// TIA Portal V18 export
// export: Created 2026-01-09T11:31:58.4430527Z, ExportSetting WithDefaults, DisplayName Totally Integrated Automation Portal, DisplayVersion V18 Update 5, DisplayName TIA Portal Openness, DisplayVersion V18 Update 5, DisplayName TIA Portal Teamcenter Gateway, DisplayVersion V18, DisplayName TIA Portal Version Control Interface, DisplayVersion V18, DisplayName SINAMICS Startdrive Advanced, DisplayVersion V18 SP2 Update 1, DisplayName SINAMICS Startdrive G110M, G120, G120C, G120D, G120P, G115D, DisplayVersion V18 SP2 Update 1, DisplayName SINAMICS Startdrive G130, G150, S120, S150, SINAMICS MV, S210, G220, S200, DisplayVersion V18 SP2 Update 1, DisplayName STEP 7 Professional, DisplayVersion V18 Update 5, DisplayName STEP 7 Safety, DisplayVersion V18, DisplayName WinCC Professional, DisplayVersion V18 Update 5
TagTable "HMI_Tool"
  ST10_RecipeDB_HMI_ParameterElement_R1GripperFixtureCode : Array [0..6] of String  (PLC tag ST10_RecipeDB_HMI.ParameterElement.R1GripperFixtureCode, CPU S71500-2PN_TP700, 1 s)
    TagArrayMember "[0]"
    TagArrayMember "[1]"
    TagArrayMember "[2]"
    TagArrayMember "[3]"
    TagArrayMember "[4]"
    TagArrayMember "[5]"
    TagArrayMember "[6]"
  ST10_RecipeDB_HMI_ParameterElement_R2GripperFixtureCode : Array [0..6] of String  (PLC tag ST10_RecipeDB_HMI.ParameterElement.R2GripperFixtureCode, CPU S71500-2PN_TP700, 1 s)
    TagArrayMember "[0]"
    TagArrayMember "[1]"
    TagArrayMember "[2]"
    TagArrayMember "[3]"
    TagArrayMember "[4]"
    TagArrayMember "[5]"
    TagArrayMember "[6]"
  ST10_RecipeDB_HMI_ParameterElement_R3GripperFixtureCode : Array [0..6] of String  (PLC tag ST10_RecipeDB_HMI.ParameterElement.R3GripperFixtureCode, CPU S71500-2PN_TP700, 1 s)
    TagArrayMember "[0]"
    TagArrayMember "[1]"
    TagArrayMember "[2]"
    TagArrayMember "[3]"
    TagArrayMember "[4]"
    TagArrayMember "[5]"
    TagArrayMember "[6]"
  ST10_RecipeDB_HMI_ParameterElement_A1RingUnloadingFixtureCode : String  (PLC tag ST10_RecipeDB_HMI.ParameterElement.A1RingUnloadingFixtureCode, CPU S71500-2PN_TP700, 1 s)
  ST10_RecipeDB_HMI_ParameterElement_E1LoadingNGFixtureCode : String  (PLC tag ST10_RecipeDB_HMI.ParameterElement.E1LoadingNGFixtureCode, CPU S71500-2PN_TP700, 1 s)
  ST10_RecipeDB_HMI_ParameterElement_ShaftScanFixtureCode : String  (PLC tag ST10_RecipeDB_HMI.ParameterElement.ShaftScanFixtureCode, CPU S71500-2PN_TP700, 1 s)
  ST10_RecipeDB_HMI_ParameterElement_B1PressFixtureCode : String  (PLC tag ST10_RecipeDB_HMI.ParameterElement.B1PressFixtureCode, CPU S71500-2PN_TP700, 1 s)
  ST10_RecipeDB_HMI_ParameterElement_CGlueFixtureCode : String  (PLC tag ST10_RecipeDB_HMI.ParameterElement.CGlueFixtureCode, CPU S71500-2PN_TP700, 1 s)
  ST10_RecipeDB_HMI_ParameterElement_B1PressCylFixtureCode : String  (PLC tag ST10_RecipeDB_HMI.ParameterElement.B1PressCylFixtureCode, CPU S71500-2PN_TP700, 1 s)
  ST10_RecipeDB_HMI_ParameterElement_A2RingUnloadingFixtureCode : String  (PLC tag ST10_RecipeDB_HMI.ParameterElement.A2RingUnloadingFixtureCode, CPU S71500-2PN_TP700, 1 s)
  ST10_RecipeDB_HMI_ParameterElement_E2UnloadingNGFixtureCode : String  (PLC tag ST10_RecipeDB_HMI.ParameterElement.E2UnloadingNGFixtureCode, CPU S71500-2PN_TP700, 1 s)
  ST10_RecipeDB_HMI_ParameterElement_B2PressFixtureCode : String  (PLC tag ST10_RecipeDB_HMI.ParameterElement.B2PressFixtureCode, CPU S71500-2PN_TP700, 1 s)
  ST10_RecipeDB_HMI_ParameterElement_CGlueNGFixtureCode : String  (PLC tag ST10_RecipeDB_HMI.ParameterElement.CGlueNGFixtureCode, CPU S71500-2PN_TP700, 1 s)
  ST10_RecipeDB_HMI_ParameterElement_B2PressCylFixtureCode : String  (PLC tag ST10_RecipeDB_HMI.ParameterElement.B2PressCylFixtureCode, CPU S71500-2PN_TP700, 1 s)
  ST10_RecipeDB_HMI_ParameterElement_A1_TableFixtureCode : Array [0..10] of String  (PLC tag ST10_RecipeDB_HMI.ParameterElement.A1_TableFixtureCode, CPU S71500-2PN_TP700, 1 s)
    TagArrayMember "[0]"
    TagArrayMember "[1]"
    TagArrayMember "[2]"
    TagArrayMember "[3]"
    TagArrayMember "[4]"
    TagArrayMember "[5]"
    TagArrayMember "[6]"
    TagArrayMember "[7]"
    TagArrayMember "[8]"
    TagArrayMember "[9]"
    TagArrayMember "[10]"
  ST10_RecipeDB_HMI_ParameterElement_A2_TableFixtureCode : Array [0..10] of String  (PLC tag ST10_RecipeDB_HMI.ParameterElement.A2_TableFixtureCode, CPU S71500-2PN_TP700, 1 s)
    TagArrayMember "[0]"
    TagArrayMember "[1]"
    TagArrayMember "[2]"
    TagArrayMember "[3]"
    TagArrayMember "[4]"
    TagArrayMember "[5]"
    TagArrayMember "[6]"
    TagArrayMember "[7]"
    TagArrayMember "[8]"
    TagArrayMember "[9]"
    TagArrayMember "[10]"
